{attribute 'linkalways'} 
{attribute 'no_explicit_call' := 'This FB is a CLASS and must be accessed using methods or properties'}
{attribute 'enable_dynamic_creation'}
FUNCTION_BLOCK _Array0to2OfSINT EXTENDS ArrayDatatypeBase_1D
VAR CONSTANT
	lBound : DINT := 0;
	uBound : DINT := 2;
END_VAR
VAR
	localData : ARRAY [lBound..uBound] OF SINT;
	activeData : REFERENCE TO ARRAY [lBound..uBound] OF SINT REF= localData;
	elements : ARRAY [lBound..uBound] OF _SINT(0);
	baseType : _SINT(0);
END_VAR

PROPERTY PUBLIC Address : PVOID
GET
Address := ADR(activeData);
END_GET
END_PROPERTY

PROPERTY PUBLIC BaseDatatype : I_Datatype
GET
BaseDatatype := baseType;
END_GET
END_PROPERTY

METHOD PUBLIC ClearReference
VAR_INPUT
END_VAR
activeData REF= localData;
SetElementReference();
END_METHOD

METHOD PUBLIC Clone : I_Datatype
VAR
    pClone : POINTER TO _Array0to2OfSINT;
END_VAR
pClone := __NEW(_Array0to2OfSINT());
pClone^.Value := Value;
Clone := pClone^;
END_METHOD

METHOD FB_init : BOOL
VAR_INPUT
	bInitRetains : BOOL; // if TRUE, the retain variables are initialized (warm start / cold start)
	bInCopyCode : BOOL;  // if TRUE, the instance afterwards gets moved into the copy code (online change)
END_VAR
SetElementReference();
END_METHOD

METHOD PUBLIC MakeReferenceTo
VAR_INPUT
	ReferenceTarget : REFERENCE TO ARRAY [lBound..uBound] OF SINT;
END_VAR
activeData REF= ReferenceTarget;
SetElementReference();
END_METHOD

METHOD PROTECTED OnSerializeArrayValues
VAR_INPUT
	Serializer : I_Serializer;
END_VAR
VAR
	i : DINT;
END_VAR
FOR i := lBound TO uBound DO
	elements[i].SerializeWith(Serializer);
END_FOR
END_METHOD

METHOD PROTECTED SetElementReference
VAR_INPUT
END_VAR
VAR
	i : DINT;
END_VAR
FOR i := lBound TO uBound DO
	elements[i].MakeReferenceTo(activeData[i]);
END_FOR
END_METHOD

PROPERTY PUBLIC Size : UDINT
GET
Size := SIZEOF(activeData);
END_GET
END_PROPERTY

METHOD PROTECTED TryDeserializeArrayValues : BOOL
VAR_INPUT
	Deserializer : I_Deserializer;
	Feedback : I_DeserializerFeedback;
END_VAR
VAR
	enumerator : I_DeserializerArrayForwardEnumerator;
	i : DINT;
END_VAR
enumerator := Deserializer.GetArrayEnumerator();
i := lBound;

WHILE enumerator.MoveNext() AND i <= uBound DO
	
	IF NOT elements[i].TryDeserializeFrom(enumerator.Current, Feedback) THEN
		EXIT;
	END_IF
	i := i + 1;

END_WHILE
enumerator.Dispose();
END_METHOD

METHOD PUBLIC TryGetElementAsDatatypeByIndex : BOOL
VAR_INPUT
	Index : DINT;
	Destination : REFERENCE TO I_Datatype;
END_VAR
IF Index < lbound OR Index > ubound THEN
	RETURN;
END_IF

Destination := elements[Index];
TryGetElementAsDatatypeByIndex := TRUE;
END_METHOD

METHOD PUBLIC TryGetLowerBound : BOOL
VAR_INPUT
	Dimention : UDINT;
	Destination : REFERENCE TO DINT;
END_VAR
IF Dimention = 1 THEN
	Destination := lBound;
	TryGetLowerBound := TRUE;
END_IF
END_METHOD

METHOD PUBLIC TryGetUpperBound : BOOL
VAR_INPUT
	Dimention : UDINT;
	Destination : REFERENCE TO DINT;
END_VAR
IF Dimention = 1 THEN
	Destination := uBound;
	TryGetUpperBound := TRUE;
END_IF
END_METHOD

METHOD TryMakeReferenceTo : BOOL
VAR_INPUT
	Target : I_Datatype;
END_VAR
VAR
	targetAsArray : I_ArrayDatatype;
	pTargetData : POINTER TO ARRAY [lBound..uBound] OF SINT;
END_VAR
IF NOT Target.TryResolveAsArrayDatatype(targetAsArray) THEN
	RETURN;
END_IF

IF NOT (targetAsArray.Identifier = Identifier) THEN
	RETURN;
END_IF

pTargetData := Target.Address;
activeData REF= pTargetData^;
SetElementReference();
TryMakeReferenceTo := TRUE;
END_METHOD

PROPERTY PUBLIC Value : REFERENCE TO ARRAY [lBound..uBound] OF SINT;
GET
Value ref= activeData;
END_GET
END_PROPERTY

END_FUNCTION_BLOCK

(* stored: Version 1.1.0.1, ProductVersion 3.1.4024.13
   POU _Array0to2OfSINT: Id {c55619c6-90b0-0c66-0884-68def61ea66b}, SpecialFunc None
   Folder Core: Id {abccc772-3238-05ba-3e51-d34a96e3ff0a}
   Folder Constructor: Id {e3ca3696-032a-030d-08b6-cf4f8238cae7}
   Folder Protected: Id {af52511c-d15a-0ca8-3b6f-4a93f77c5614}
   Folder Customize: Id {1057c5be-8783-0225-0058-073e9e140800}
   Property Address: Id {929ef1b8-a103-09c4-1a4e-03a385bc4e5a}
   Get Get: Id {b2fa3fd5-9840-0938-18f6-d7c92ea59acf}
   Property BaseDatatype: Id {96d5e600-b8fd-0a1b-3de5-bfa572ffe581}
   Get Get: Id {0cb9451e-b485-09d9-1430-4c2374d0eb75}
   Method ClearReference: Id {ec83d813-fba2-0a4c-112e-192231c283a4}
   Method Clone: Id {ac210812-aa30-0850-0a89-51eb18f0e966}
   Method FB_init: Id {88d1659e-b00a-0000-1a0f-e607ce422ea0}
   Method MakeReferenceTo: Id {de6a87e4-bd0e-0b55-172b-9fed302b6e5c}
   Method OnSerializeArrayValues: Id {ae277c73-3db6-0f37-3ea0-b82dd61a4f51}
   Method SetElementReference: Id {683cf2ef-05f7-07cc-2a51-402711b4a43a}
   Property Size: Id {2bcab1d3-f4e6-0c4b-0276-eb6a41b687a7}
   Get Get: Id {043678e3-ccb4-00d2-0f99-ef23122c9ee1}
   Method TryDeserializeArrayValues: Id {5c253547-2650-0772-1d89-24857d1b0b7b}
   Method TryGetElementAsDatatypeByIndex: Id {de7af8c8-f3ba-0744-3b20-d78ffd931cbd}
   Method TryGetLowerBound: Id {9c03ffc0-abce-0315-372b-92c016352bc2}
   Method TryGetUpperBound: Id {cf527cec-a091-0b52-3115-ef94b5a08118}
   Method TryMakeReferenceTo: Id {b027183a-ac07-03ee-2212-6d133f7a0625}
   Property Value: Id {2dca74fe-e280-0532-1736-c719f386e9c4}
   Get Get: Id {e6d8aa93-68ac-044b-341b-34c2785e5d01} *)
